// TIA Portal project "conveyer belt system V4.2" (V19)

(* hardware
DEVICE "S71500/ET200MP-Station_1"  S7-1500 station
   slot 0: "Profilschiene_0"  6ES7 590-1***0-0AA0
   slot 1: "PLC_1"  CPU 1511-1 PN  6ES7 511-1AK00-0AB0  V1.8
   slot 2: "AI 8xU/I/RTD/TC ST_1"  AI 8xU/I/RTD/TC ST  6ES7 531-7KF00-0AB0  V2.0
   slot 3: "AI 8xU/I/RTD/TC ST_2"  AI 8xU/I/RTD/TC ST  6ES7 531-7KF00-0AB0  V2.0
   slot 4: "AI 8xU/I/RTD/TC ST_3"  AI 8xU/I/RTD/TC ST  6ES7 531-7KF00-0AB0  V2.0
   slot 5: "AI 8xU/I/RTD/TC ST_4"  AI 8xU/I/RTD/TC ST  6ES7 531-7KF00-0AB0  V2.0
   slot 6: "DI 16x24VDC BA_1"  DI 16x24VDC BA  6ES7 521-1BH10-0AA0  V1.0
*)

// ===== PLC "PLC_1"  CPU 1511-1 PN =====

VAR_GLOBAL   // PLC tag table "Standard-Variablentabelle"
   "Tag_1" AT %I1000.0 : Bool;
   "Tag_2" AT %Q1000.0 : Bool;
   "Tag_3" AT %I1000.1 : Bool;
END_VAR

VAR_GLOBAL   // PLC tag table "control panel"
   "start button" AT %I0.0 : Bool;
   "reset button" AT %I0.1 : Bool;
   "stop button" AT %I0.2 : Bool;
   "emergency stop" AT %I0.3 : Bool;
   "start button light" AT %Q0.0 : Bool;
   "reset button light" AT %Q0.1 : Bool;
   "stop button light" AT %Q0.2 : Bool;
   "system start" AT %Q0.3 : Bool;
   "system fault" AT %Q0.4 : Bool;
   "system stop" AT %Q0.5 : Bool;
   "sensor start" AT %I4.0 : Bool;
   "low power mode" AT %I0.4 : Bool;
END_VAR

VAR_GLOBAL   // PLC tag table "conveyor 0"
   "motor +(0)" AT %Q3.7 : Bool;
   "motor -(0)" AT %Q3.6 : Bool;
   "encoder A(0)" AT %I2.7 : Bool;
   "encoder B(0)" AT %I2.6 : Bool;
   "sensor(0)" AT %I3.7 : Bool;
END_VAR

VAR_GLOBAL   // PLC tag table "conveyor 1"
   "motor +(1)" AT %Q3.5 : Bool;
   "motor -(1)" AT %Q3.4 : Bool;
   "encoder A(1)" AT %I2.5 : Bool;
   "encoder B(1)" AT %I2.4 : Bool;
   "sensor(1)" AT %I3.6 : Bool;
END_VAR

VAR_GLOBAL   // PLC tag table "conveyor 2"
   "motor +(2)" AT %Q3.3 : Bool;
   "motor -(2)" AT %Q3.2 : Bool;
   "encoder A(2)" AT %I2.2 : Bool;
   "encoder B(2)" AT %I2.3 : Bool;
   "sensor(2)" AT %I3.5 : Bool;
END_VAR

VAR_GLOBAL   // PLC tag table "system state"
   "start 0" AT %M0.0 : Bool;
   "start 1" AT %M0.1 : Bool;
   "conveyor 2 running" AT %M10.2 : Bool;
   "conveyor 1 running" AT %M10.1 : Bool;
   "conveyor 0 running" AT %M10.0 : Bool;
   "sensor 0 memory" AT %M20.0 : Bool;
   "sensor 1 memory" AT %M20.1 : Bool;
   "sensor 2 memory" AT %M20.2 : Bool;
   "sensor start memory" AT %M30.0 : Bool;
   "all conveyors running" AT %M0.2 : Bool;
   "system start/stop memory" AT %M0.4 : Bool;
   "conveyors running" AT %M0.3 : Bool;
END_VAR

DATA_BLOCK "conveyor_0"   // DB1
{ S7_Optimized_Access := 'TRUE' }
VERSION : 0.1
// stored: InstanceOfName conveyor
"conveyor"
BEGIN
END_DATA_BLOCK

DATA_BLOCK "conveyor_2"   // DB3
{ S7_Optimized_Access := 'TRUE' }
VERSION : 0.1
// stored: InstanceOfName conveyor
"conveyor"
BEGIN
END_DATA_BLOCK

DATA_BLOCK "conveyor_1"   // DB5
{ S7_Optimized_Access := 'TRUE' }
VERSION : 0.1
// stored: InstanceOfName conveyor
"conveyor"
BEGIN
END_DATA_BLOCK

DATA_BLOCK "sensor control_0"   // DB8
{ S7_Optimized_Access := 'TRUE' }
VERSION : 0.1
// stored: InstanceOfName sensor control
"sensor control"
BEGIN
END_DATA_BLOCK

DATA_BLOCK "sensor control_1"   // DB9
{ S7_Optimized_Access := 'TRUE' }
VERSION : 0.1
// stored: InstanceOfName sensor control
"sensor control"
BEGIN
END_DATA_BLOCK

DATA_BLOCK "sensor control_2"   // DB10
{ S7_Optimized_Access := 'TRUE' }
VERSION : 0.1
// stored: InstanceOfName sensor control
"sensor control"
BEGIN
END_DATA_BLOCK

DATA_BLOCK "lamp control_DB"   // DB11
{ S7_Optimized_Access := 'TRUE' }
VERSION : 0.1
// stored: InstanceOfName lamp control
"lamp control"
BEGIN
END_DATA_BLOCK

DATA_BLOCK "start pulse"   // DB12
{ S7_Optimized_Access := 'TRUE' }
VERSION : 0.1
// stored: InstanceOfName pulse
"pulse"
BEGIN
END_DATA_BLOCK

DATA_BLOCK "stop pulse"   // DB13
{ S7_Optimized_Access := 'TRUE' }
VERSION : 0.1
// stored: InstanceOfName pulse
"pulse"
BEGIN
END_DATA_BLOCK

// folder: System blocks/Program resources

DATA_BLOCK "conveyor start delay"   // DB2
{ S7_Optimized_Access := 'TRUE' }
AUTHOR : Simatic
FAMILY : IEC
NAME : IEC_TMR
VERSION : 1.0
// stored: InstanceOfName IEC_TIMER
"IEC_TIMER"
BEGIN
END_DATA_BLOCK

DATA_BLOCK "delay 1"   // DB4
{ S7_Optimized_Access := 'TRUE' }
AUTHOR : Simatic
FAMILY : IEC
NAME : IEC_TMR
VERSION : 1.0
// stored: InstanceOfName IEC_TIMER
"IEC_TIMER"
BEGIN
END_DATA_BLOCK

DATA_BLOCK "delay 2"   // DB6
{ S7_Optimized_Access := 'TRUE' }
AUTHOR : Simatic
FAMILY : IEC
NAME : IEC_TMR
VERSION : 1.0
// stored: InstanceOfName IEC_TIMER
"IEC_TIMER"
BEGIN
END_DATA_BLOCK

DATA_BLOCK "delay 0"   // DB7
{ S7_Optimized_Access := 'TRUE' }
AUTHOR : Simatic
FAMILY : IEC
NAME : IEC_TMR
VERSION : 1.0
// stored: InstanceOfName IEC_TIMER
"IEC_TIMER"
BEGIN
END_DATA_BLOCK

// folder: (top level)

FUNCTION_BLOCK "conveyor"   // FB1, FBD
{ S7_Optimized_Access := 'TRUE' }
VERSION : 0.1
   VAR_INPUT
      enable : Bool;
      "encoder A" : Bool;
      "encoder B" : Bool;
      "clearance time" : Time := T#500MS;
   END_VAR
   VAR_OUTPUT
      "running feedback" : Bool;
      "motor +" : Bool;
      "motor -" : Bool;
   END_VAR
   VAR
      "encoder buffer" : TOF_TIME;
      "encoder A edge" : R_TRIG;
      "encoder B edge" : R_TRIG;
   END_VAR
BEGIN

REGION Network 1
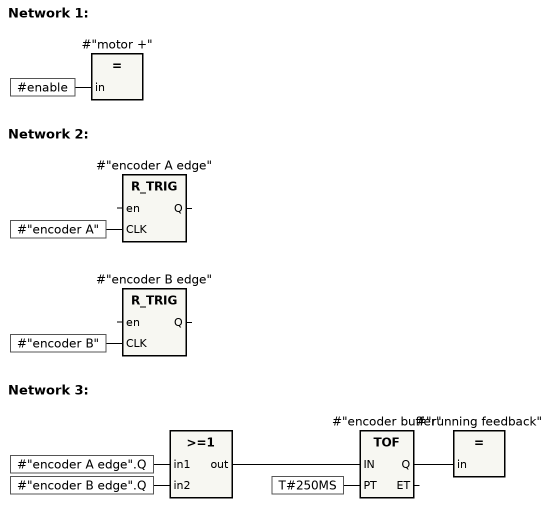
   #"motor +" := #enable;
END_REGION

REGION Network 2
   #"encoder A edge"(CLK := #"encoder A");   // R_TRIG
   #"encoder B edge"(CLK := #"encoder B");   // R_TRIG
END_REGION

REGION Network 3
   #"encoder buffer"(IN := #"encoder A edge".Q OR #"encoder B edge".Q, PT := T#250MS);   // TOF
   #"running feedback" := #"encoder buffer".Q;
END_REGION
END_FUNCTION_BLOCK

FUNCTION_BLOCK "sensor control"   // FB2, FBD
{ S7_Optimized_Access := 'TRUE' }
VERSION : 0.1
   VAR_INPUT
      "clearance time" : Time;
      sensor : Bool;
      "preceding sensor" : Bool;
   END_VAR
   VAR_OUTPUT
      "motor +" : Bool;
   END_VAR
   VAR_IN_OUT
      "sensor memory" : Bool;
   END_VAR
   VAR
      "clearance timer off" : TOF_TIME;
      "clearance timer on" : TOF_TIME;
   END_VAR
BEGIN

REGION Network 1
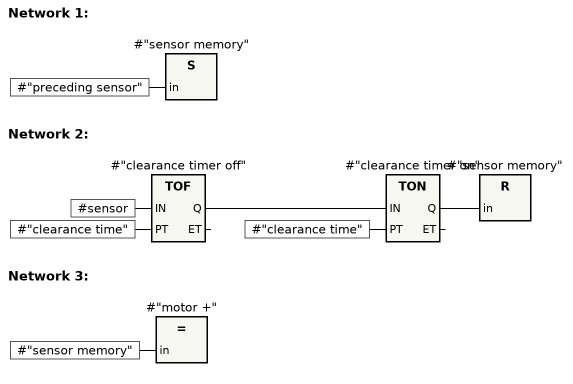
   IF #"preceding sensor" THEN #"sensor memory" := TRUE; END_IF;
END_REGION

REGION Network 2
   #"clearance timer off"(IN := #sensor, PT := #"clearance time");   // TOF
   #"clearance timer on"(IN := #"clearance timer off".Q, PT := #"clearance time");   // TON
   IF #"clearance timer on".Q THEN #"sensor memory" := FALSE; END_IF;
END_REGION

REGION Network 3
   #"motor +" := #"sensor memory";
END_REGION
END_FUNCTION_BLOCK

FUNCTION_BLOCK "lamp control"   // FB3, FBD
{ S7_Optimized_Access := 'TRUE' }
VERSION : 0.1
   VAR_INPUT
      "system start" : Bool;
      "system fault" : Bool;
      "system stop" : Bool;
   END_VAR
BEGIN

REGION Network 1
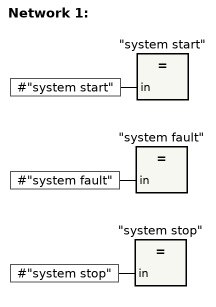
   "system start" := #"system start";
   "system fault" := #"system fault";
   "system stop" := #"system stop";
END_REGION
END_FUNCTION_BLOCK

FUNCTION_BLOCK "pulse"   // FB4, FBD
{ S7_Optimized_Access := 'TRUE' }
VERSION : 0.1
   VAR_INPUT
      enable : Bool;
      "pulse time" : Time;
   END_VAR
   VAR_OUTPUT
      "pulsing output" : Bool;
   END_VAR
   VAR
      "time delay bit" : Bool;
      IEC_Timer_0_Instance : TON_TIME;
      IEC_Timer_0_Instance_1 : TON_TIME;
   END_VAR
BEGIN

REGION Network 1
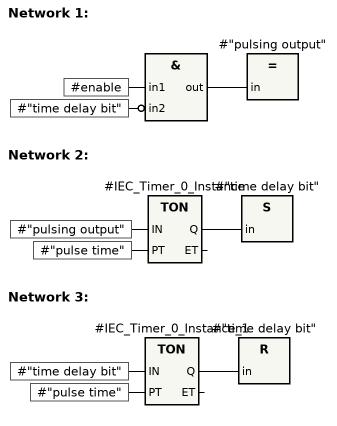
   #"pulsing output" := #enable AND NOT #"time delay bit";
END_REGION

REGION Network 2
   #IEC_Timer_0_Instance(IN := #"pulsing output", PT := #"pulse time");   // TON
   IF #IEC_Timer_0_Instance.Q THEN #"time delay bit" := TRUE; END_IF;
END_REGION

REGION Network 3
   #IEC_Timer_0_Instance_1(IN := #"time delay bit", PT := #"pulse time");   // TON
   IF #IEC_Timer_0_Instance_1.Q THEN #"time delay bit" := FALSE; END_IF;
END_REGION
END_FUNCTION_BLOCK

FUNCTION "default condition" : Void   // FC1, FBD
{ S7_Optimized_Access := 'TRUE' }
VERSION : 0.1
   VAR_INPUT
      "clearance delay" : Time;
      "low power clearance delay" : Time;
      "pulse time" : Time;
   END_VAR
   VAR_TEMP   // added for the SCL form of the ladder/FBD networks
      _w1 : Bool;
      _w2 : Bool;
      _w3 : Bool;
   END_VAR
BEGIN

REGION Network 1
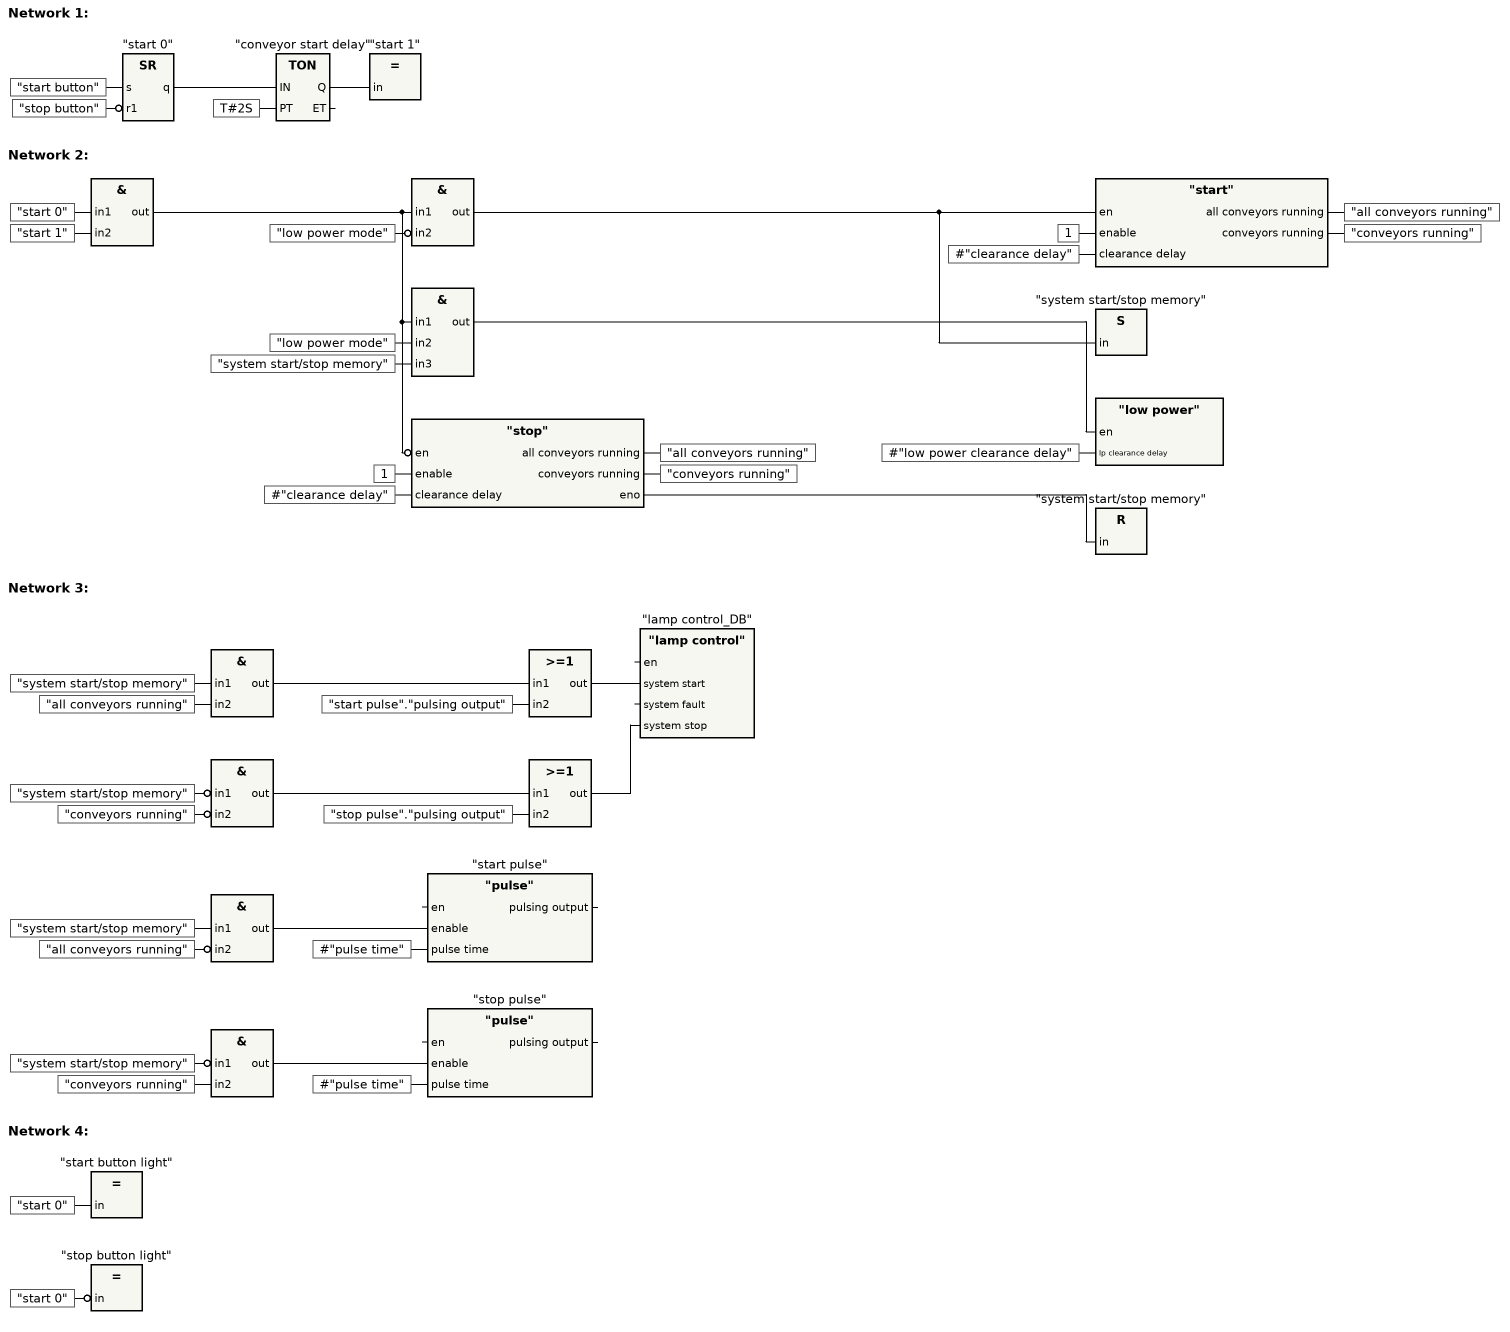
   IF "start button" THEN
       "start 0" := TRUE;   // SR flip-flop
   END_IF;
   IF NOT "stop button" THEN "start 0" := FALSE; END_IF;
   "conveyor start delay".TON(IN := "start 0", PT := T#2S);
   "start 1" := "conveyor start delay".Q;
END_REGION

REGION Network 2
   #_w1 := "start 0" AND "start 1";
   #_w2 := #_w1 AND NOT "low power mode";
   IF #_w2 THEN
       "start"(enable := 1,
               "clearance delay" := #"clearance delay",
               "all conveyors running" => "all conveyors running",
               "conveyors running" => "conveyors running");
       "system start/stop memory" := TRUE;
   END_IF;
   IF #_w1 AND "low power mode" AND "system start/stop memory" THEN
       "low power"("lp clearance delay" := #"low power clearance delay");
   END_IF;
   "stop"(EN := NOT #_w1,
          enable := 1,
          "clearance delay" := #"clearance delay",
          "all conveyors running" => "all conveyors running",
          "conveyors running" => "conveyors running",
          ENO => #_w3);
   IF #_w3 THEN "system start/stop memory" := FALSE; END_IF;
END_REGION

REGION Network 3
   "lamp control_DB"("system start" := ("system start/stop memory" AND "all conveyors running") OR "start pulse"."pulsing output",   // "lamp control"
                     "system stop" := (NOT "system start/stop memory" AND NOT "conveyors running") OR "stop pulse"."pulsing output");
   "start pulse"(enable := "system start/stop memory" AND NOT "all conveyors running",   // "pulse"
                 "pulse time" := #"pulse time");
   "stop pulse"(enable := NOT "system start/stop memory" AND "conveyors running", "pulse time" := #"pulse time");   // "pulse"
END_REGION

REGION Network 4
   "start button light" := "start 0";
   "stop button light" := NOT "start 0";
END_REGION
END_FUNCTION

FUNCTION "start" : Void   // FC2, FBD
{ S7_Optimized_Access := 'TRUE' }
VERSION : 0.1
   VAR_INPUT
      enable : Bool;
      "clearance delay" : Time;
   END_VAR
   VAR_OUTPUT
      "all conveyors running" : Bool;
      "conveyors running" : Bool;
   END_VAR
BEGIN

REGION Network 1
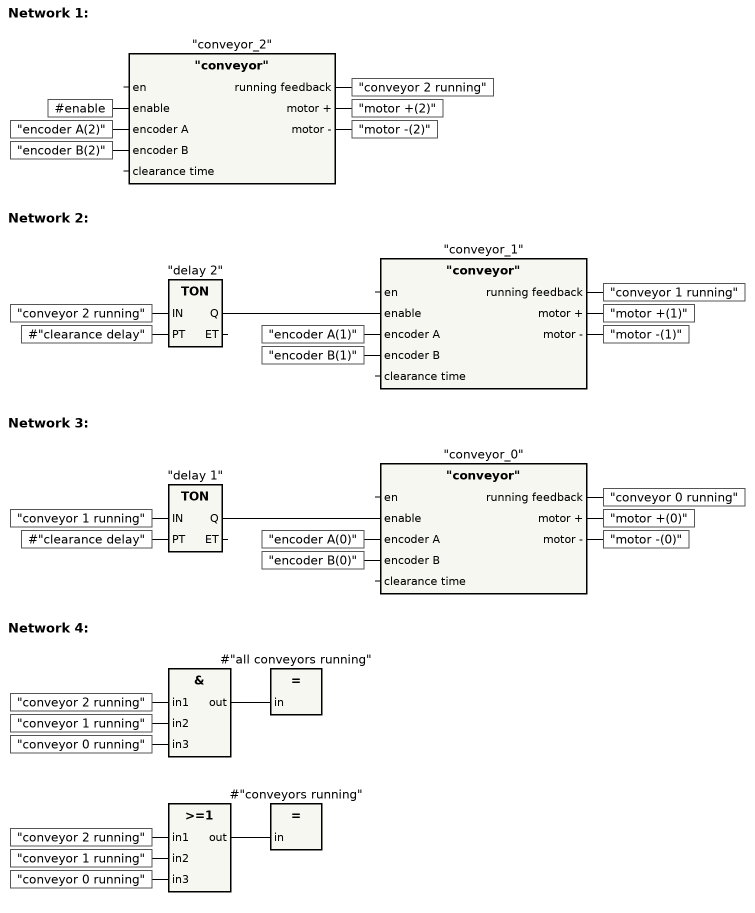
   "conveyor_2"(enable := #enable,   // "conveyor"
                "encoder A" := "encoder A(2)",
                "encoder B" := "encoder B(2)",
                "running feedback" => "conveyor 2 running",
                "motor +" => "motor +(2)",
                "motor -" => "motor -(2)");
END_REGION

REGION Network 2
   "delay 2".TON(IN := "conveyor 2 running", PT := #"clearance delay");
   "conveyor_1"(enable := "delay 2".Q,   // "conveyor"
                "encoder A" := "encoder A(1)",
                "encoder B" := "encoder B(1)",
                "running feedback" => "conveyor 1 running",
                "motor +" => "motor +(1)",
                "motor -" => "motor -(1)");
END_REGION

REGION Network 3
   "delay 1".TON(IN := "conveyor 1 running", PT := #"clearance delay");
   "conveyor_0"(enable := "delay 1".Q,   // "conveyor"
                "encoder A" := "encoder A(0)",
                "encoder B" := "encoder B(0)",
                "running feedback" => "conveyor 0 running",
                "motor +" => "motor +(0)",
                "motor -" => "motor -(0)");
END_REGION

REGION Network 4
   #"all conveyors running" := "conveyor 2 running" AND "conveyor 1 running" AND "conveyor 0 running";
   #"conveyors running" := "conveyor 2 running" OR "conveyor 1 running" OR "conveyor 0 running";
END_REGION
END_FUNCTION

FUNCTION "stop" : Void   // FC3, FBD
{ S7_Optimized_Access := 'TRUE' }
VERSION : 0.1
   VAR_INPUT
      enable : Bool;
      "clearance delay" : Time;
   END_VAR
   VAR_OUTPUT
      "all conveyors running" : Bool;
      "conveyors running" : Bool;
   END_VAR
BEGIN

REGION Network 1
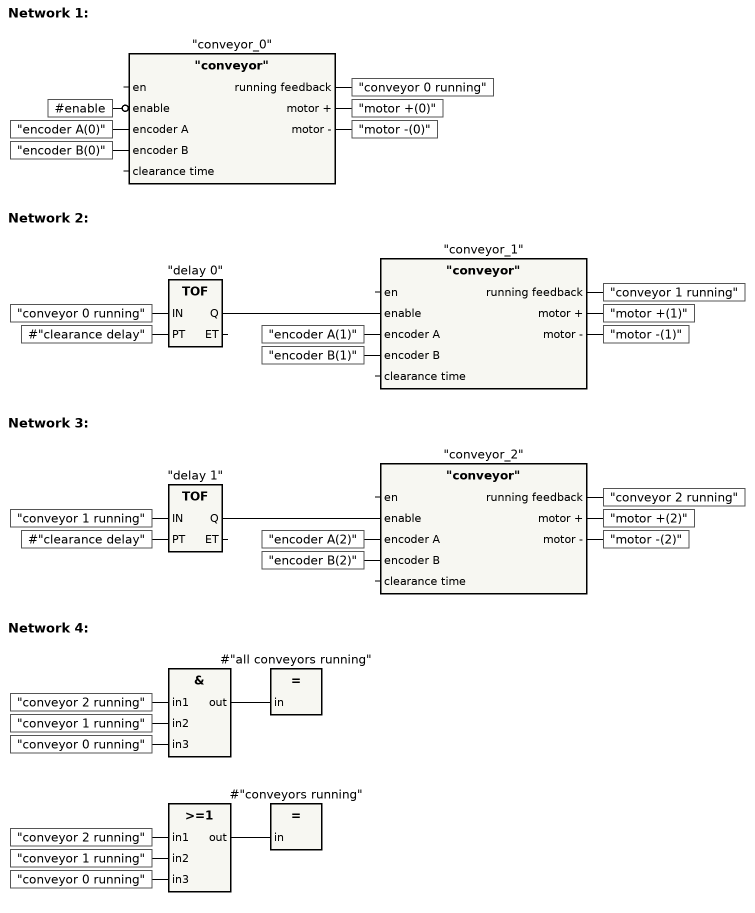
   "conveyor_0"(enable := NOT #enable,   // "conveyor"
                "encoder A" := "encoder A(0)",
                "encoder B" := "encoder B(0)",
                "running feedback" => "conveyor 0 running",
                "motor +" => "motor +(0)",
                "motor -" => "motor -(0)");
END_REGION

REGION Network 2
   "delay 0".TOF(IN := "conveyor 0 running", PT := #"clearance delay");
   "conveyor_1"(enable := "delay 0".Q,   // "conveyor"
                "encoder A" := "encoder A(1)",
                "encoder B" := "encoder B(1)",
                "running feedback" => "conveyor 1 running",
                "motor +" => "motor +(1)",
                "motor -" => "motor -(1)");
END_REGION

REGION Network 3
   "delay 1".TOF(IN := "conveyor 1 running", PT := #"clearance delay");
   "conveyor_2"(enable := "delay 1".Q,   // "conveyor"
                "encoder A" := "encoder A(2)",
                "encoder B" := "encoder B(2)",
                "running feedback" => "conveyor 2 running",
                "motor +" => "motor +(2)",
                "motor -" => "motor -(2)");
END_REGION

REGION Network 4
   #"all conveyors running" := "conveyor 2 running" AND "conveyor 1 running" AND "conveyor 0 running";
   #"conveyors running" := "conveyor 2 running" OR "conveyor 1 running" OR "conveyor 0 running";
END_REGION
END_FUNCTION

FUNCTION "low power" : Void   // FC4, FBD
{ S7_Optimized_Access := 'TRUE' }
VERSION : 0.1
   VAR_INPUT
      "lp clearance delay" : Time;
   END_VAR
   VAR_TEMP   // added for the SCL form of the ladder/FBD networks
      _w1 : Bool;
   END_VAR
BEGIN

REGION Network 1
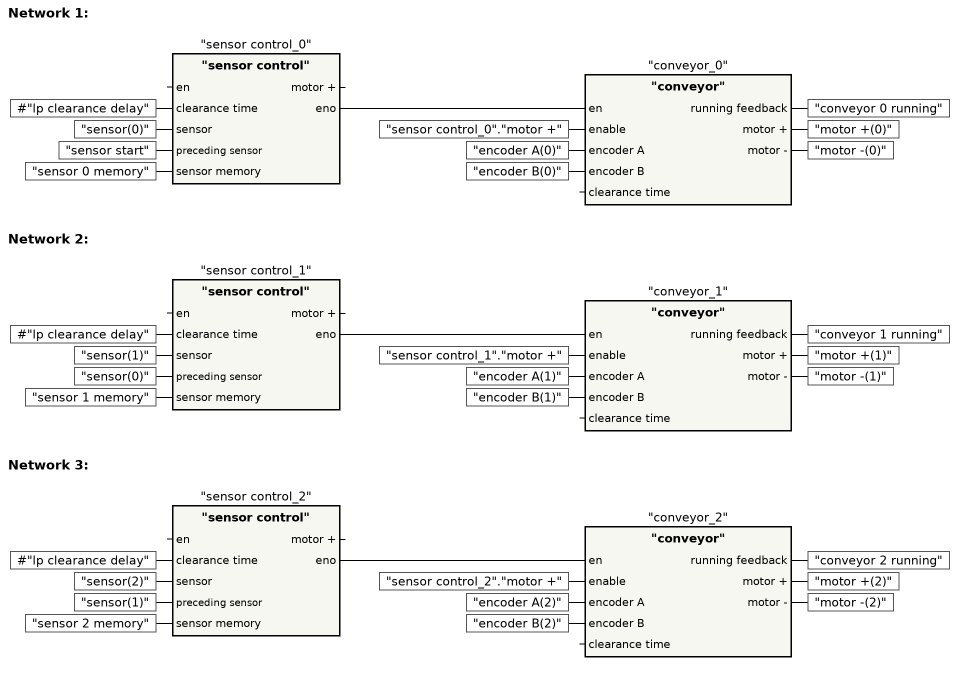
   "sensor control_0"("clearance time" := #"lp clearance delay",   // "sensor control"
                      sensor := "sensor(0)",
                      "preceding sensor" := "sensor start",
                      "sensor memory" := "sensor 0 memory",
                      ENO => #_w1);
   IF #_w1 THEN
       "conveyor_0"(enable := "sensor control_0"."motor +",   // "conveyor"
                    "encoder A" := "encoder A(0)",
                    "encoder B" := "encoder B(0)",
                    "running feedback" => "conveyor 0 running",
                    "motor +" => "motor +(0)",
                    "motor -" => "motor -(0)");
   END_IF;
END_REGION

REGION Network 2
   "sensor control_1"("clearance time" := #"lp clearance delay",   // "sensor control"
                      sensor := "sensor(1)",
                      "preceding sensor" := "sensor(0)",
                      "sensor memory" := "sensor 1 memory",
                      ENO => #_w1);
   IF #_w1 THEN
       "conveyor_1"(enable := "sensor control_1"."motor +",   // "conveyor"
                    "encoder A" := "encoder A(1)",
                    "encoder B" := "encoder B(1)",
                    "running feedback" => "conveyor 1 running",
                    "motor +" => "motor +(1)",
                    "motor -" => "motor -(1)");
   END_IF;
END_REGION

REGION Network 3
   "sensor control_2"("clearance time" := #"lp clearance delay",   // "sensor control"
                      sensor := "sensor(2)",
                      "preceding sensor" := "sensor(1)",
                      "sensor memory" := "sensor 2 memory",
                      ENO => #_w1);
   IF #_w1 THEN
       "conveyor_2"(enable := "sensor control_2"."motor +",   // "conveyor"
                    "encoder A" := "encoder A(2)",
                    "encoder B" := "encoder B(2)",
                    "running feedback" => "conveyor 2 running",
                    "motor +" => "motor +(2)",
                    "motor -" => "motor -(2)");
   END_IF;
END_REGION
END_FUNCTION

FUNCTION "MHJ-PLC-Lab-Function-S71500" : Void   // FC9000, SCL
{ S7_Optimized_Access := 'TRUE' }
VERSION : 0.1
   VAR_TEMP
      Value : Byte;
      ForCounter : Int;
   END_VAR
   VAR CONSTANT
      Value_01_DW : DWord := 16#1223_5486;
      Value_02_DW : DWord := 16#A6C9_D1F5;
   END_VAR
BEGIN

   #Value:=PEEK(area := 16#82,
        dbNumber := 0,
        byteOffset := 511);
   #Value := #Value + 1;

   POKE(area := 16#82,
        dbNumber := 0,
        byteOffset := 511,
        value := #Value);

   POKE(area := 16#82,
        dbNumber := 0,
        byteOffset := 1016,
        value := #Value_01_DW);
   POKE(area := 16#82,
        dbNumber := 0,
        byteOffset := 1020,
        value := #Value_02_DW);

   FOR #ForCounter := 0 TO 63 DO
       #Value:=PEEK(area := 16#1,
            dbNumber := 0,
            byteOffset := #ForCounter);
       POKE(area := 16#81,
            dbNumber := 0,
            byteOffset := #ForCounter,
            value := #Value);
   END_FOR;
   #Value := PEEK(area := 16#1,
                  dbNumber := 0,
                  byteOffset := 512);
   POKE(area := 16#82,
        dbNumber := 0,
        byteOffset := 512,
        value := #Value);
END_FUNCTION

ORGANIZATION_BLOCK "Main"   // OB1, FBD, ProgramCycle
TITLE = "Main Program Sweep (Cycle)"
{ S7_Optimized_Access := 'TRUE' }
VERSION : 0.1
   VAR_INPUT
      Initial_Call : Bool;   // Initial call of this OB
      Remanence : Bool;   // =True, if remanent data are available
   END_VAR
BEGIN

REGION Network 1
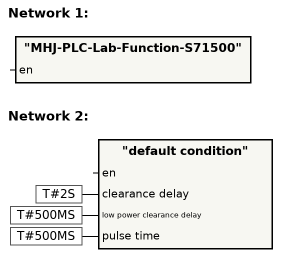
   "MHJ-PLC-Lab-Function-S71500"();
END_REGION

REGION Network 2
   "default condition"("clearance delay" := T#2S,
                       "low power clearance delay" := T#500MS,
                       "pulse time" := T#500MS);
END_REGION
END_ORGANIZATION_BLOCK